FUNCTION_BLOCK F_MIN (* minimum *)
  (* Standard: 61131-3; Classification: standard selection function *)
  (* Version 1.0, 2011-09-28, 4DIAC-IDE, 4DIAC-Consortium *)
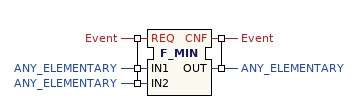
  EVENT_INPUT
    REQ WITH IN1, IN2; (* Service Request *)
  END_EVENT
  EVENT_OUTPUT
    CNF WITH OUT; (* Confirmation of Requested Service *)
  END_EVENT
  VAR_INPUT
    IN1 : ANY_ELEMENTARY; (* Input value 1 *)
    IN2 : ANY_ELEMENTARY; (* Input value 2 *)
  END_VAR
  VAR_OUTPUT
    OUT : ANY_ELEMENTARY; (* Minimum value *)
  END_VAR
END_FUNCTION_BLOCK
